(* CODESYS project image_32_Bit_xLH_base_lernpfad_pneumatik_vps_sps_01_00.project
   Description: Receives some incoming messages and echoes them with CAN-ID +1
   Author: 3S - Smart Software Solutions GmbH
   Version: 1.0.0.0
   Title: CAN Bus API Example
   Company: 3S - Smart Software Solutions GmbH

Project tree, tasks and I/O mapping:
  XLH_base : CODESYS Control for Raspberry Pi SL, CODESYS, order no. 2302000009, version 4.12.0.0
    application app
      libraries: Standard, 3.5.18.0 (System); Memory, * (3S - Smart Software Solutions GmbH); Util, 3.5.19.0 (System); VisuDialogs, * (System); CAA Tick Extern, 3.5.17.0 (CAA Technical Workgroup); SysTime, 3.5.17.0 (System); CmpIecTask, * (System); SysTypes Interfaces, * (System); SysShm, * (System); xemax Bibliothek, 0.20 (xemax ag); Memory, 3.5.17.0 (3S - Smart Software Solutions GmbH)
      task MAIN_TASK (cyclic, interval 20 ms, priority 0) calls MAIN, io, io_fs
      task VISU_TASK (cyclic, interval 100 ms, priority 31) calls VisuElems.Visu_Prg
      task RGB_TASK (cyclic, interval 20 ms, priority 10) calls XLH_RGB
      Symbols
      visualisation VISU
      program MAIN [ST]
      io/
        program io [ST]
        program io_fs [ST]: in, out
        program XLH_RGB [ST]
      program DAUERZYKLUS_ST [ST]
      program DAUERZYKLUS_FUP [FBD]
      Hinweise/
        fluidsim
        RNDIS_Driver
    SoftMotion General Axis Pool
    GPIOs_A_B : GPIOs B+/Pi2, CODESYS, version 4.12.0.0
        input  app.io.bSw1 : BOOL  // digital inputs (GPIO0..GPIO31).Bit4
        input  app.io.bSw2 : BOOL  // digital inputs (GPIO0..GPIO31).Bit5
        input  app.io.bSw3 : BOOL  // digital inputs (GPIO0..GPIO31).Bit6
        input  app.io.bSw4 : BOOL  // digital inputs (GPIO0..GPIO31).Bit12
        input  app.io.bSw5 : BOOL  // digital inputs (GPIO0..GPIO31).Bit13
        input  app.io.bSw6 : BOOL  // digital inputs (GPIO0..GPIO31).Bit16
        input  app.io.bSw7 : BOOL  // digital inputs (GPIO0..GPIO31).Bit17
        input  app.io.bSw8 : BOOL  // digital inputs (GPIO0..GPIO31).Bit19
        output app.io.bLed1 : BOOL  // digital outputs (GPIO0..GPIO31).Bit20
        output app.io.bLed2 : BOOL  // digital outputs (GPIO0..GPIO31).Bit21
        output app.io.bLed3 : BOOL  // digital outputs (GPIO0..GPIO31).Bit22
        output app.io.bLed4 : BOOL  // digital outputs (GPIO0..GPIO31).Bit23
        output app.io.bLed5 : BOOL  // digital outputs (GPIO0..GPIO31).Bit24
        output app.io.bLed6 : BOOL  // digital outputs (GPIO0..GPIO31).Bit26
        output app.io.bLed7 : BOOL  // digital outputs (GPIO0..GPIO31).Bit27
        unmapped channels: digital inputs (GPIO0..GPIO31), digital outputs (GPIO0..GPIO31)
    Onewire
    Camera device
      <Leer>
    SPI
    I²C
    Ethernet : Ethernet, CODESYS, version 4.2.0.0
        settings: IPAddress = [127,0,0,1]; SubnetMask = [255,0,0,0]; GatewayAddress = [0,0,0,0]; NetworkInterfaceName = 'lo'; NetworkInterfaceName = "lo"; SaveCommunicationSettings = FALSE
      ModbusTCP_Slave_OLED_Port_503 : ModbusTCP Slave Device, CODESYS, version 4.3.0.0
          settings: Port = 503
          output app.io.oled.awToOled : ARRAY[0..32] OF WORD  // Ausgänge
          unmapped channels: Eingänge
  libraries: VisuSymbols, 4.5.0.0 (System); DepictorBase, 1.0.5.0 (3S - Smart Software Solutions GmbH)
  text list GlobalTextList
  text list System
  00000000-0000-0000-0000-000000000000|E:\xemax ag\prj_24_03_xLH - Allgemein\Image\RNDIS_Driver.zip
*)

// XLH_base/app/MAIN
PROGRAM MAIN
VAR
	vVersionPlc: VERSION;
	sVersionPlc: STRING(255);
	vVersionLib: VERSION;
	sVersionLib: STRING(255);
	
	bFluidsim_S1: BOOL;
	bDummy: bool;
END_VAR

// Version Bibliothex xemax
vVersionPlc.uiMajor := 1;
vVersionPlc.uiMinor := 0;
sVersionPlc := CONCAT(TO_STRING(TO_UINT(vVersionPlc.uiMajor)), CONCAT('.', (TO_STRING(TO_UINT(vVersionPlc.uiMinor)))));
vVersionLib := xemax.GetLibVersion();
sVersionLib := CONCAT(TO_STRING(TO_UINT(vVersionLib.uiMajor)), CONCAT('.', (TO_STRING(TO_UINT(vVersionLib.uiMinor)))));

// Lernpfad Pneumatik - VPS - SPS
io_fs.in();// lesen der Eingänge Fluidsim

DAUERZYKLUS_FUP();
DAUERZYKLUS_ST();

io_fs.out();// schreiben der Ausgänge Fluidsim


bDummy := bFluidsim_S1;


(*
==================================================================================================
Login Codesys in die XLH - SPS 
user: pi
pw: pi
==================================================================================================
Webvisualisierung
http://ip:8080/webvisu.htm
- bei einer Verbindung via USB: http://192.168.31.31:8080/webvisu.htm
- bei einer Verbindung via USB-RJ45-Adapter: http://192.168.1.31:8080/webvisu.htm
==================================================================================================
OPC-UA
anonymous (ohne Benutzer und Passwort)
opc.tcp://192.168.31.31:4840
==================================================================================================
RGB-Matrix
im aktuellen BETA-Status kann die Matrix via REST-API angesteurt werden
https://de.wikipedia.org/wiki/Representational_State_Transfer
http://192.168.1.31:8077/rgb/0/1/0

Weiter geplant ist eine Umsetzung zur Ansteuerung der RGB Matrix als IoT Device via MQTT
 
Die Integration in Codesys ist noch ausstehend 
==================================================================================================
Login XLH - Linuxumgebung via Putty
user: pi
pw: pi
==================================================================================================
Konfiguration WiFi 
sudo nano /etc/wpa_supplicant/wpa_supplicant.conf

network={
        ssid="abc"
        psk="def"
        key_mgmt=WPA-PSK
}
==================================================================================================
statische IP USB-Ethernet-Erweiterung: 
sudo nano /etc/dhcpcd.conf
# profile static_eth0
...
==================================================================================================
*)

END_PROGRAM

// XLH_base/app/io/io_fs
PROGRAM io_fs
VAR_INPUT
	byFluidsimIn: BYTE;
	//
	bY1: BOOL;
	bY2: BOOL;
	bFsOut2: BOOL;
	bFsOut3: BOOL;
	bFsOut4: BOOL;
	bFsOut5: BOOL;
	bFsOut6: BOOL;
	bFsOut7: BOOL;	
END_VAR
VAR_OUTPUT
	byFluidsimOut: UINT;
	//
	bS1: BOOL;
	bS2: BOOL;
	bS3: BOOL;
	bB1: BOOL;
	bB2: BOOL;
	bFsIn5: BOOL;
	bFsIn6: BOOL;
	bFsIn7: BOOL;
END_VAR
VAR
	fbUnpackByte: MEM.UnpackByte;	
END_VAR

// siehe auch YouTube https://www.youtube.com/watch?v=EhQRrw3T-Is

{region}
//https://www.codesys.com/fileadmin/data/News_Images/good-to-know/CODESYS-video-ST-code-via-Pragma.mp4
{endregion}

ACTION in:
// Byte nach 8 x BOOL
fbUnpackByte(byValue := TO_BYTE(byFluidsimIn));	
bS1 := fbUnpackByte.xBit0;
bS2 := fbUnpackByte.xBit1;
bS3 := fbUnpackByte.xBit2;
bB1 := fbUnpackByte.xBit3;
bB2 := fbUnpackByte.xBit4;
bFsIn5 := fbUnpackByte.xBit5;
bFsIn6 := fbUnpackByte.xBit6;
bFsIn7 := fbUnpackByte.xBit7;
END_ACTION

ACTION out:
// 8 x BOOL nach Byte
byFluidsimOut := MEM.PackBitsToByte(
	bFsOut7,
	bFsOut6,
	bFsOut5,
	bFsOut4,
	bFsOut3,
	bFsOut2,
	bY2,
	bY1);
END_ACTION

END_PROGRAM

// XLH_base/app/DAUERZYKLUS_FUP
PROGRAM DAUERZYKLUS_FUP
VAR_OUTPUT
	fbTonB2: TON;
END_VAR
VAR
	bEnable: BOOL;	
	fbSrEnable: SR;
	fbSrY1: SR;
	fbSrY2: SR;
END_VAR

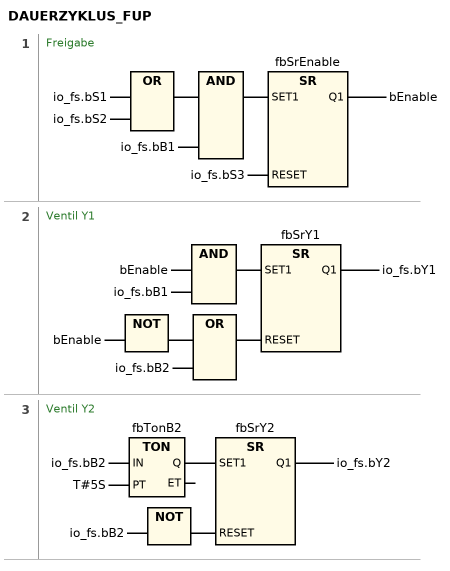
// NETWORK 1
// Freigabe
fbSrEnable(SET1 := (io_fs.bS1 OR io_fs.bS2) AND io_fs.bB1, RESET := io_fs.bS3); // SR
bEnable := fbSrEnable.Q1;

// NETWORK 2
// Ventil Y1
fbSrY1(SET1 := bEnable AND io_fs.bB1, RESET := NOT bEnable OR io_fs.bB2); // SR
io_fs.bY1 := fbSrY1.Q1;

// NETWORK 3
// Ventil Y2
fbTonB2(IN := io_fs.bB2, PT := T#5S); // TON
fbSrY2(SET1 := fbTonB2.Q, RESET := NOT io_fs.bB2); // SR
io_fs.bY2 := fbSrY2.Q1;

END_PROGRAM

// XLH_base/app/DAUERZYKLUS_ST
PROGRAM DAUERZYKLUS_ST
VAR
	bEnable: BOOL;	
	fbTonB2: TON;
END_VAR

// siehe auch YouTube https://www.youtube.com/watch?v=EhQRrw3T-Is

(*
// Logikprogrammierung in ST
IF io_fs.bS1 OR io_fs.bS2 THEN
	bEnable := TRUE;
END_IF
IF io_fs.bS3 THEN
	bEnable := FALSE;
END_IF

IF io_fs.bB1 AND bEnable THEN
	io_fs.bY1 := TRUE;
END_IF
IF io_fs.bB2 OR NOT bEnable THEN
	io_fs.bY1 := FALSE;
END_IF

fbTonB2(IN:=io_fs.bB2, PT:=T#5S);
IF fbTonB2.Q THEN
	io_fs.bY2 := TRUE;
END_IF
IF NOT io_fs.bB2 THEN
	io_fs.bY2 := FALSE;
END_IF
*)



// Anzeige der Endschalter und Ventile auf dem xLH_base
io.bLed1 := io_fs.bB1;
io.bLed2 := io_fs.bB2;
// RGB 8x8 Ausgabe der Ventilzustände
IF io_fs.bY1 THEN
	io.rgb[0,0].byRed := 0;
	io.rgb[0,0].byGreen := 25;
ELSE
	io.rgb[0,0].byRed := 50;
	io.rgb[0,0].byGreen := 0;
END_IF
IF io_fs.bY2 THEN
	io.rgb[0,7].byRed := 0;
	io.rgb[0,7].byGreen := 25;
ELSE
	io.rgb[0,7].byRed := 50;
	io.rgb[0,7].byGreen := 0;
END_IF
	 
// Anzeige OLED
io.oled.bShowLines := io.bSw4;
io.oled.sLine1.sText := 'Lernpfad';
io.oled.sLine2.sText := 'Pneumatik';
io.oled.sLine3.sText := 'SPS xLH';
io.oled.sLine4.sText := 'TON: ';
io.oled.sLine4.sText := CONCAT(io.oled.sLine4.sText, 
                               TO_STRING(TO_LREAL(DAUERZYKLUS_FUP.fbTonB2.ET)/1000.0));
io.oled.sLine4.sText := CONCAT(io.oled.sLine4.sText, ' s');

END_PROGRAM

// XLH_base/app/io/io
PROGRAM io
VAR_INPUT			
	bLed1: BOOL;
	bLed2: BOOL;
	bLed3: BOOL;
	bLed4: BOOL;
	bLed5: BOOL;
	bLed6: BOOL;
	bLed7: BOOL;	
	oled: xemax.OLED;
	rgb: ARRAY[0..7, 0..7] OF xemax.RGB_PIXEL;
END_VAR
VAR_OUTPUT
	bSw1: BOOL;
	bSw2: BOOL;
	bSw3: BOOL;
	bSw4: BOOL;
	bSw5: BOOL;
	bSw6: BOOL;
	bSw7: BOOL;
	bSw8: BOOL;
END_VAR
VAR
END_VAR

xemax.LOCAL_TIME_AND_TIME_ZONE();
xemax.TASK_INFO();
oled();

END_PROGRAM

// XLH_base/app/io/XLH_RGB
PROGRAM XLH_RGB
VAR
END_VAR

xemax.RGB_SHARED_MEMORY(bEnable:=io.bSw4, rgb:=io.rgb);

END_PROGRAM

// XLH_base/app/VISU
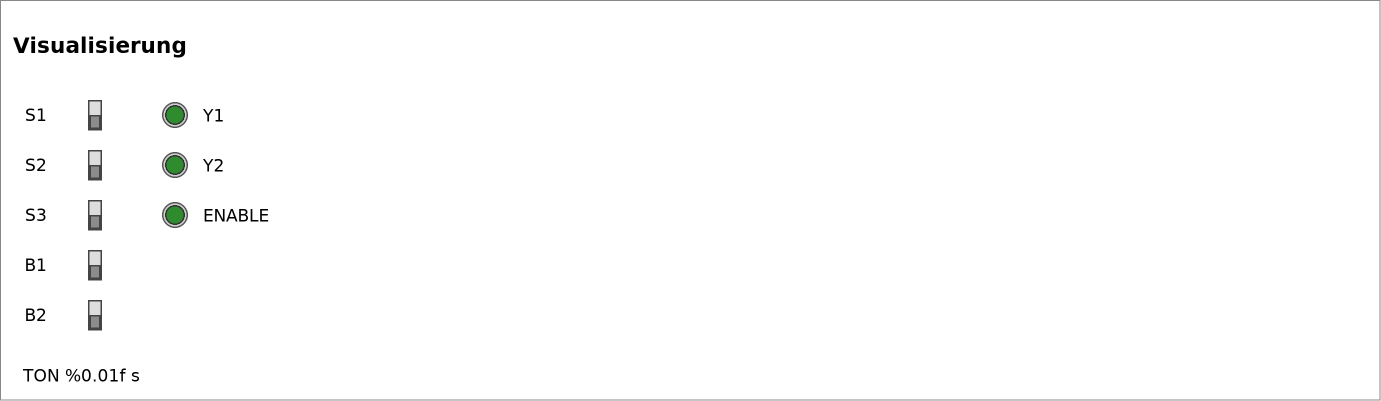
VISUALIZATION VISU  // 1381x401
    Rectangle (200,90 81x51), "Y1"
    Rectangle (10,10 271x71), "Visualisierung"
    Line (1380,270)
    DipSwitch (60,100 70x30), variable: io_fs.bS1, behaviour: TOGGLE, style: Switch-DipSwitch-Gray
    Rectangle (0,90 50x50), "S1"
    Lamp1 (160,100 30x30), variable: io_fs.bY1, style: Lamp-Lamp1-Green
    Rectangle (0,140 50x50), "S2"
    DipSwitch (60,150 70x30), variable: io_fs.bS2, behaviour: TOGGLE, style: Switch-DipSwitch-Gray
    Rectangle (200,140 81x51), "Y2"
    DipSwitch (60,200 70x30), variable: io_fs.bS3, behaviour: TOGGLE, style: Switch-DipSwitch-Gray
    Rectangle (0,190 50x50), "S3"
    Lamp1 (160,150 30x30), variable: io_fs.bY2, style: Lamp-Lamp1-Green
    Rectangle (0,240 50x50), "B1"
    DipSwitch (60,250 70x30), variable: io_fs.bB1, behaviour: TOGGLE, style: Switch-DipSwitch-Gray
    DipSwitch (60,300 70x30), variable: io_fs.bB2, behaviour: TOGGLE, style: Switch-DipSwitch-Gray
    Rectangle (0,290 50x50), "B2"
    Rectangle (20,350 191x51), "TON %0.01f s", text variable: TO_LREAL(DAUERZYKLUS_FUP.fbTonB2.ET) / 1000.0
    Rectangle (200,190 91x51), "ENABLE"
    Lamp1 (160,200 30x30), variable: DAUERZYKLUS_FUP.bEnable, style: Lamp-Lamp1-Green
END_VISUALIZATION

(* text list System (id | default)
  Apr | Apr
  April | April
  Aug | Aug
  August | August
  Dec | Dec
  December | December
  Feb | Feb
  February | February
  Fri | Fri
  Friday | Friday
  Jan | Jan
  January | January
  Jul | Jul
  July | July
  Jun | Jun
  June | June
  Mar | Mar
  March | March
  May | May
  May_3Letter | May
  Mon | Mon
  Monday | Monday
  Nov | Nov
  November | November
  Oct | Oct
  October | October
  Sat | Sat
  Saturday | Saturday
  Sep | Sep
  September | September
  Sun | Sun
  Sunday | Sunday
  Thu | Thu
  Thursday | Thursday
  Tue | Tue
  Tuesday | Tuesday
  Wed | Wed
  Wednesday | Wednesday
   |  *)
